Universal Robots URScript: Test Square Motion.script

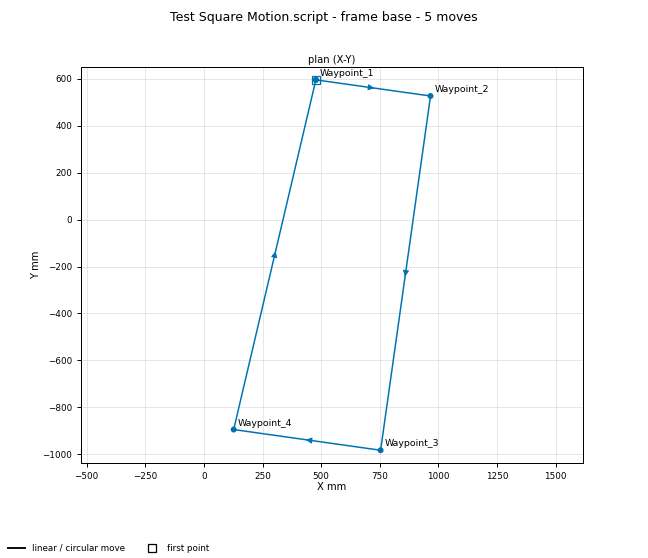
[picture p0: tool path of Test Square Motion.script in frame base, 5 of 5 moves have a stored position in this frame; points joined in program order, loops and branches not executed]
def Test_Square_Motion():
  global _hidden_verificationVariable=0
  set_standard_analog_input_domain(0, 1)
  set_standard_analog_input_domain(1, 1)
  set_tool_analog_input_domain(0, 1)
  set_tool_analog_input_domain(1, 1)
  set_analog_outputdomain(0, 0)
  set_analog_outputdomain(1, 0)
  set_input_actions_to_default()
  set_target_payload(1.130000, [0.000000, 0.003000, 0.000000], [0.001887, 0.001887, 0.001887, 0.000000, 0.000000, 0.000000])
  set_safety_mode_transition_hardness(1)
  set_gravity([0.0, 0.0, 9.82])
  set_tool_communication(False, 115200, 0, 1, 1.5, 3.5)
  set_tool_output_mode(0)
  set_tool_digital_output_mode(0, 1)
  set_tool_digital_output_mode(1, 1)
  set_tool_voltage(0)
  set_tcp(p[-4.516483728619642E-6,-4.494070941040221E-6,-3.385497268221845E-5,0.0,0.0,0.0])
  # begin: URCap Installation Node
  #   Source: MachineLogic for Universal Robots, 3.1.7, Vention Inc.
  #   Type: MachineLogic for Universal Robots
  def waitForResponse(expected_response_vention, cname_vention):
  response_vention = socket_read_string(cname_vention,timeout=15)
  while response_vention != expected_response_vention:
  sleep(0.01)
  response_vention = socket_read_string(cname_vention,timeout=15)
  end
  sleep(0.01)
  sync()
  end
  def sendString(string_vention, expected_response_vention, cname_vention):
  socket_send_string(str_cat(string_vention,";"), cname_vention)
  response_vention = socket_read_string(cname_vention,timeout=15)
  if(response_vention == "nAck"):
  popup("nAck received")
  end
  while response_vention != expected_response_vention:
  sleep(0.01)
  response_vention = socket_read_string(cname_vention,timeout=15)
  if(response_vention == "nAck"):
  popup("nAck received")
  end
  end
  sleep(0.01)
  sync()
  end
  def sendStringNAck(string_vention, expected_response_vention, cname_vention):
  socket_send_string(str_cat(string_vention,";"), cname_vention)
  response_vention = socket_read_string(cname_vention,timeout=15)
  if(response_vention == "nAck"):
  popup("nAck received")
  end
  while(response_vention != expected_response_vention and response_vention != "nAck"):
  sleep(0.01)
  response_vention = socket_read_string(cname_vention,timeout=15)
  if(response_vention == "nAck"):
  popup("nAck received",blocking=True)
  end
  end
  sleep(0.01)
  sync()
  end
  def sendStringWithTimeout(string_vention, expected_response_vention, cname_vention):
  socket_send_string(str_cat(string_vention,";"), cname_vention)
  response_vention = socket_read_string(cname_vention,timeout=10)
  if(response_vention == "nAck"):
  popup("nAck received"+string_vention)
  end
  sleep(0.01)
  sync()
  end
  def pollString(string_vention, expected_response_vention, cname_vention):
  socket_send_string(str_cat(string_vention,";"), cname_vention)
  response_vention = socket_read_string(cname_vention,timeout=15)
  if(response_vention == "nAck"):
  popup("nAck received")
  end
  while response_vention != expected_response_vention:
  sleep(1)
  socket_send_string(str_cat(string_vention,";"), cname_vention)
  response_vention = socket_read_string(cname_vention,timeout=15)
  if(response_vention == "nAck"):
  popup("nAck received")
  end
  end
  sleep(0.01)
  sync()
  end
  def sendVariable(var_vention, data_vention, expected_response_vention, cname_vention):
  socket_set_var(var_vention, data_vention, cname_vention)
  response_vention = socket_read_string(cname_vention,timeout=15)
  if(response_vention == "nAck"):
  popup("nAck received")
  end
  while response_vention != expected_response_vention:
  sleep(0.01)
  response_vention = socket_read_string(cname_vention,timeout=15)
  if(response_vention == "nAck"):
  popup("nAck received")
  end
  end
  sleep(0.01)
  sync()
  end
  def intToString(integer_vention,cname_vention):
  stringFix=""
  multiplier_vention123=1
  if integer_vention<0:
  stringFix="-"
  multiplier_vention123=-1
  end
  socket_set_var("GetString",integer_vention*multiplier_vention123,cname_vention)
  string_vention=""
  while string_vention=="":
  sleep(0.01)
  string_vention=socket_read_string(cname_vention,timeout=15)
  end
  sleep(0.01)
  sync()
  string_vention=stringFix+string_vention
  return string_vention
  end
  string_vention=""
  isVentionMovementBusy = False
  isVentionParallelMovementSendingScript = False
  ventionThreadHandle = 1
  isVentionMovementBusyMachineMotion1 = False
  isVentionParallelMovementSendingScriptMachineMotion1 = False
  socket_vention = socket_open("192.168.7.2", 9999, "MachineMotion1")
  if socket_vention==False:
  popup("Check configuration, can't connect to MachineMotion")
  end
  waitForResponse("MachineMotion connection established", "MachineMotion1")
  sendString("isReady", "MachineMotion isReady = true", "MachineMotion1")
  sendStringWithTimeout("setURCapVersion2", "setURCapVersion loaded", "MachineMotion1")
  sendString("SET speed_v2 1000000", "Ack", "MachineMotion1")
  sendString("SET acceleration_v2 100000", "Ack", "MachineMotion1")
  sendString("SET de_axis_1_microsteps_config 8", "Ack", "MachineMotion1")
  sendString("SET de_axis_1_mechanical_gain_config_v2 150000.0", "Ack", "MachineMotion1")
  sendString("SET de_axis_1_direction_config 1", "Ack", "MachineMotion1")
  sendString("SET de_axis_1_type_config Electric Cylinder ", "Ack", "MachineMotion1")
  sendString("de_axis_1_config_exec", "Ack", "MachineMotion1")
  # end: URCap Installation Node
  step_count_b08da966_eb90_4c2b_a80f_05093ec7b23c = 0.0
  thread Step_Counter_Thread_d50d775c_67fa_4c0f_b85a_8a6ec00c00a3():
    while (True):
      step_count_b08da966_eb90_4c2b_a80f_05093ec7b23c = step_count_b08da966_eb90_4c2b_a80f_05093ec7b23c + 1.0
      sync()
    end
  end
  run Step_Counter_Thread_d50d775c_67fa_4c0f_b85a_8a6ec00c00a3()
  global Waypoint_1_p=p[.477467448927, .596236493009, .273466520488, -1.989451343072, 2.359750942138, .026824631245]
  global Waypoint_1_q=[1.162696123123169, -1.847117086450094, -2.3881099224090576, -0.4209882777980347, 1.5623012781143188, 1.3325953483581543]
  global Waypoint_2_p=p[.966474445477, .527332164483, .273447487952, -1.989455373213, 2.359772914978, .026776961290]
  global Waypoint_2_q=[0.6797319054603577, -2.113852163354391, -1.895011305809021, -0.6497024458697815, 1.5899512767791748, 0.850642204284668]
  global Waypoint_3_p=p[.753568009387, -.983519102738, .273449564694, -1.989463101915, 2.359782412820, .026765185087]
  global Waypoint_3_q=[-0.7618635336505335, -2.229412694970602, -1.6476792097091675, -0.8473634284785767, 1.6280813217163086, -0.5917308966266077]
  global Waypoint_4_p=p[.126889569685, -.895203556087, .273464202366, -1.989490200116, 2.359771979032, .026734180429]
  global Waypoint_4_q=[-1.2146404425250452, -1.9531051121153773, -2.1635663509368896, -0.6313834947398682, 1.6172142028808594, -1.0452821890460413]
  while (True):
    $ 2 "Robot Program"
    $ 3 "MoveL"
    $ 4 "Waypoint_1" "breakAfter"
    movel(Waypoint_1_p, a=1.2, v=0.25)
    $ 5 "Waypoint_2" "breakAfter"
    movel(Waypoint_2_p, a=1.2, v=0.25)
    $ 6 "Waypoint_3" "breakAfter"
    movel(Waypoint_3_p, a=1.2, v=0.25)
    $ 7 "Waypoint_4" "breakAfter"
    movel(Waypoint_4_p, a=1.2, v=0.25)
    $ 8 "Waypoint_1" "breakAfter"
    movel(Waypoint_1_p, a=1.2, v=0.25)
  end
end
